PROGRAM MAIN
VAR
	bFlag			:BOOL;
END_VAR

GVL_General.myTimer.Delay(in:=T#5S);

IF	GVL_General.myTimer.bDone THEN 
	bFlag := TRUE;
	
	
END_IF

END_PROGRAM

(* stored: Version 1.1.0.1, ProductVersion 3.1.4022.16
   POU MAIN: Id {ccb61117-473d-422a-b215-ba03d30bcee5}, SpecialFunc None *)
